% RSLogix 500 project LADDER LOGIC OF INTERLOCK CIRCUIT_BAK013.RSS, saved by version 8.30.00.16 %
PROJECT "UNTITLED"    % processor: Bul.1763 MicroLogix 1100 Series B %

PROGRAM FILES
  LAD 2   7 rungs

DATA FILES
  O0 OUTPUT  4 elements
  I1 INPUT  6 elements
  S2 STATUS  66 elements
  B3 BINARY  1 elements
  T4 TIMER  1 elements
  C5 COUNTER  1 elements
  R6 CONTROL  1 elements
  N7 INTEGER  1 elements
  F8 FLOAT  1 elements

LADDER 2
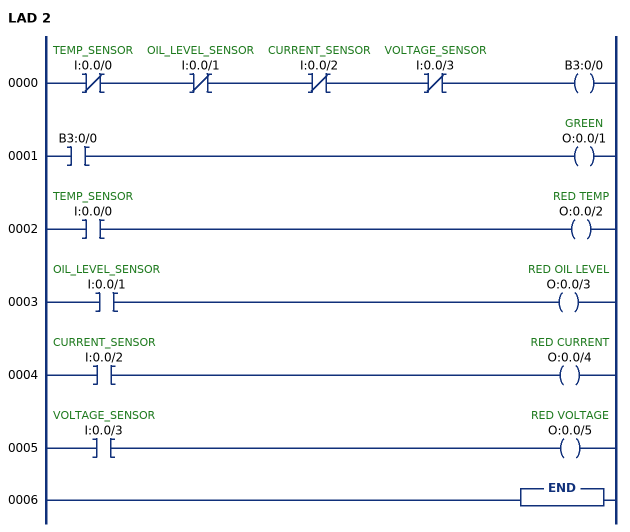
% Rung: 0 %
SOR XIO I:0.0/0 XIO I:0.0/1 XIO I:0.0/2 XIO I:0.0/3 OTE B3:0/0 EOR
%   I:0.0/0  TEMP_SENSOR %
%   I:0.0/1  OIL_LEVEL_SENSOR %
%   I:0.0/2  CURRENT_SENSOR %
%   I:0.0/3  VOLTAGE_SENSOR %
% Rung: 1 %
SOR XIC B3:0/0 OTE O:0.0/1 EOR
%   O:0.0/1  "GREEN" %
% Rung: 2 %
SOR XIC I:0.0/0 OTE O:0.0/2 EOR
%   I:0.0/0  TEMP_SENSOR %
%   O:0.0/2  "RED TEMP" %
% Rung: 3 %
SOR XIC I:0.0/1 OTE O:0.0/3 EOR
%   I:0.0/1  OIL_LEVEL_SENSOR %
%   O:0.0/3  "RED OIL LEVEL" %
% Rung: 4 %
SOR XIC I:0.0/2 OTE O:0.0/4 EOR
%   I:0.0/2  CURRENT_SENSOR %
%   O:0.0/4  "RED CURRENT" %
% Rung: 5 %
SOR XIC I:0.0/3 OTE O:0.0/5 EOR
%   I:0.0/3  VOLTAGE_SENSOR %
%   O:0.0/5  "RED VOLTAGE" %
% Rung: 6 %
SOR END EOR

OTHER DOCUMENTED ADDRESSES
  O:0.0/0  DISPLAY
